FUNCTION_BLOCK TON_Mock_TimerRanOut IMPLEMENTS I_TON
VAR_INPUT
END_VAR
VAR_OUTPUT
END_VAR
VAR
    _mockQ : BOOL := TRUE;
    _mockET : TIME := T#0S;
END_VAR

 
METHOD Call : BOOL
VAR_INPUT
	IN	: BOOL;
	PT	: TIME;
END_VAR
VAR_OUTPUT
	Q : BOOL;
	ET : TIME;
END_VAR
// Simulate timer behavior for unit testing
IF IN THEN
	_mockQ := TRUE;  // Simulate timer has finished
ELSE
	_mockQ := FALSE;
END_IF
_mockET := PT;  // Pretend elapsed time matches preset
Q := _mockQ;
ET := _mockET;
END_METHOD

END_FUNCTION_BLOCK

(* stored: Version 1.1.0.1, ProductVersion 3.1.4024.9
   POU TON_Mock_TimerRanOut: Id {e4eaacbd-35c4-4076-9dfd-55b2686f215b}, SpecialFunc None
   Method Call: Id {838dc7fc-3948-44ca-b936-b6c5d5e25610} *)
